(* PLC project static_torsion.project, CODESYS CODESYS V3.5 SP17 Patch 3 *)
(* stored: creationDateTime 1970-01-01T00:00:00, modificationDateTime 2026-06-22T15:12:39.4699931 *)

TYPE REAL_WORD2 : UNION
  _REAL : REAL;
  _WORDS : ARRAY[0..1] OF WORD;
END_UNION;
END_TYPE
